Fanuc TP program (LS listing): DISTI_CADC_V16.LS

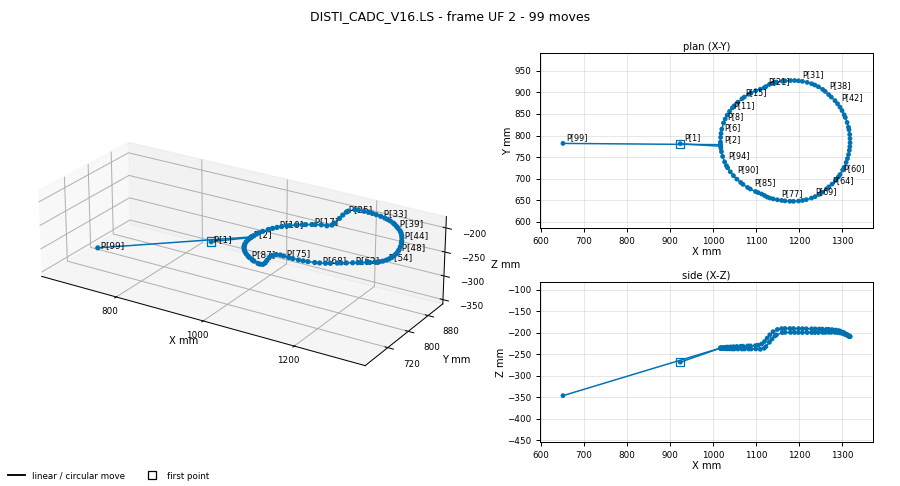
[picture p0: tool path of DISTI_CADC_V16.LS in frame UF 2, 99 of 99 moves have a stored position in this frame; points joined in program order, loops and branches not executed]
/PROG  DISTI_CADC_V16
/ATTR
OWNER		= MNEDITOR;
COMMENT		= "WeldPRO Auto-Gen";
PROG_SIZE	= 7125;
CREATE		= DATE 26-07-30  TIME 16:10:00;
MODIFIED	= DATE 26-07-30  TIME 16:41:22;
FILE_NAME	= DISTI_CA;
VERSION		= 0;
LINE_COUNT	= 113;
MEMORY_SIZE	= 7445;
PROTECT		= READ_WRITE;
TCD:  STACK_SIZE	= 0,
      TASK_PRIORITY	= 50,
      TIME_SLICE	= 0,
      BUSY_LAMP_OFF	= 0,
      ABORT_REQUEST	= 0,
      PAUSE_REQUEST	= 0;
DEFAULT_GROUP	= 1,*,*,*,*;
CONTROL_CODE	= 00000000 00000000;
/APPL
/MN
   1:  !WeldPRO Auto-Generated TPP ;
   2:  !TOR_XL_2026, TOR_xl_2907 ;
   3:   ;
   4:  UFRAME_NUM=2 ;
   5:  UTOOL_NUM=2 ;
   6:  !Feature Approach ;
   7:J P[1] 100% FINE    ;
   8:   ;
   9:  !Segment1 ;
  10:L P[2] 2000mm/sec FINE    ;
  11:   ;
  12:  CALL LASER_OFF    ;
  13:L P[3] R[23:moving]mm/sec CNT100    ;
  14:L P[4] R[23:moving]mm/sec CNT100    ;
  15:L P[5] R[23:moving]mm/sec CNT100    ;
  16:L P[6] R[23:moving]mm/sec CNT100    ;
  17:L P[7] R[23:moving]mm/sec CNT100    ;
  18:L P[8] R[23:moving]mm/sec CNT100    ;
  19:L P[9] R[23:moving]mm/sec CNT100    ;
  20:L P[10] R[23:moving]mm/sec CNT100    ;
  21:L P[11] R[23:moving]mm/sec CNT100    ;
  22:L P[12] R[23:moving]mm/sec CNT100    ;
  23:L P[13] R[23:moving]mm/sec CNT100    ;
  24:L P[14] R[23:moving]mm/sec CNT100    ;
  25:L P[15] R[23:moving]mm/sec CNT100    ;
  26:L P[16] R[23:moving]mm/sec CNT100    ;
  27:L P[17] R[23:moving]mm/sec CNT100    ;
  28:L P[18] R[23:moving]mm/sec CNT100    ;
  29:L P[19] R[23:moving]mm/sec CNT100    ;
  30:L P[20] R[23:moving]mm/sec CNT100    ;
  31:L P[21] R[23:moving]mm/sec CNT100    ;
  32:L P[22] R[23:moving]mm/sec CNT100    ;
  33:L P[23] R[23:moving]mm/sec CNT100    ;
  34:L P[24] R[23:moving]mm/sec CNT100    ;
  35:L P[25] R[23:moving]mm/sec CNT100    ;
  36:L P[26] R[23:moving]mm/sec CNT100    ;
  37:L P[27] R[23:moving]mm/sec CNT100    ;
  38:L P[28] R[23:moving]mm/sec CNT100    ;
  39:L P[29] R[23:moving]mm/sec CNT100    ;
  40:L P[30] R[23:moving]mm/sec CNT100    ;
  41:L P[31] R[23:moving]mm/sec CNT100    ;
  42:L P[32] R[23:moving]mm/sec CNT100    ;
  43:L P[33] R[23:moving]mm/sec CNT100    ;
  44:L P[34] R[23:moving]mm/sec CNT100    ;
  45:L P[35] R[23:moving]mm/sec CNT100    ;
  46:L P[36] R[23:moving]mm/sec CNT100    ;
  47:L P[37] R[23:moving]mm/sec CNT100    ;
  48:L P[38] R[23:moving]mm/sec CNT100    ;
  49:L P[39] R[23:moving]mm/sec CNT100    ;
  50:L P[40] R[23:moving]mm/sec CNT100    ;
  51:L P[41] R[23:moving]mm/sec CNT100    ;
  52:L P[42] R[23:moving]mm/sec CNT100    ;
  53:L P[43] R[23:moving]mm/sec CNT100    ;
  54:L P[44] R[23:moving]mm/sec CNT100    ;
  55:L P[45] R[23:moving]mm/sec CNT100    ;
  56:L P[46] R[23:moving]mm/sec CNT100    ;
  57:L P[47] R[23:moving]mm/sec CNT100    ;
  58:L P[48] R[23:moving]mm/sec CNT100    ;
  59:L P[49] R[23:moving]mm/sec CNT100    ;
  60:L P[50] R[23:moving]mm/sec CNT100    ;
  61:L P[51] R[23:moving]mm/sec CNT100    ;
  62:L P[52] R[23:moving]mm/sec CNT100    ;
  63:L P[53] R[23:moving]mm/sec CNT100    ;
  64:L P[54] R[23:moving]mm/sec CNT100    ;
  65:L P[55] R[23:moving]mm/sec CNT100    ;
  66:L P[56] R[23:moving]mm/sec CNT100    ;
  67:L P[57] R[23:moving]mm/sec CNT100    ;
  68:L P[58] R[23:moving]mm/sec CNT100    ;
  69:L P[59] R[23:moving]mm/sec CNT100    ;
  70:L P[60] R[23:moving]mm/sec CNT100    ;
  71:L P[61] R[23:moving]mm/sec CNT100    ;
  72:L P[62] R[23:moving]mm/sec CNT100    ;
  73:L P[63] R[23:moving]mm/sec CNT100    ;
  74:L P[64] R[23:moving]mm/sec CNT100    ;
  75:L P[65] R[23:moving]mm/sec CNT100    ;
  76:L P[66] R[23:moving]mm/sec CNT100    ;
  77:L P[67] R[23:moving]mm/sec CNT100    ;
  78:L P[68] R[23:moving]mm/sec CNT100    ;
  79:L P[69] R[23:moving]mm/sec CNT100    ;
  80:L P[70] R[23:moving]mm/sec CNT100    ;
  81:L P[71] R[23:moving]mm/sec CNT100    ;
  82:L P[72] R[23:moving]mm/sec CNT100    ;
  83:L P[73] R[23:moving]mm/sec CNT100    ;
  84:L P[74] R[23:moving]mm/sec CNT100    ;
  85:L P[75] R[23:moving]mm/sec CNT100    ;
  86:L P[76] R[23:moving]mm/sec CNT100    ;
  87:L P[77] R[23:moving]mm/sec CNT100    ;
  88:L P[78] R[23:moving]mm/sec CNT100    ;
  89:L P[79] R[23:moving]mm/sec CNT100    ;
  90:L P[80] R[23:moving]mm/sec CNT100    ;
  91:L P[81] R[23:moving]mm/sec CNT100    ;
  92:L P[82] R[23:moving]mm/sec CNT100    ;
  93:L P[83] R[23:moving]mm/sec CNT100    ;
  94:L P[84] R[23:moving]mm/sec CNT100    ;
  95:L P[85] R[23:moving]mm/sec CNT100    ;
  96:L P[86] R[23:moving]mm/sec CNT100    ;
  97:L P[87] R[23:moving]mm/sec CNT100    ;
  98:L P[88] R[23:moving]mm/sec CNT100    ;
  99:L P[89] R[23:moving]mm/sec CNT100    ;
 100:L P[90] R[23:moving]mm/sec CNT100    ;
 101:L P[91] R[23:moving]mm/sec CNT100    ;
 102:L P[92] R[23:moving]mm/sec CNT100    ;
 103:L P[93] R[23:moving]mm/sec CNT100    ;
 104:L P[94] R[23:moving]mm/sec CNT100    ;
 105:L P[95] R[23:moving]mm/sec CNT100    ;
 106:L P[96] R[23:moving]mm/sec CNT100    ;
 107:L P[97] R[23:moving]mm/sec CNT100    ;
 108:L P[98] R[23:moving]mm/sec FINE    ;
 109:  CALL LASER_OFF    ;
 110:   ;
 111:  !Feature Retreat ;
 112:L P[99] 2000mm/sec FINE    ;
 113:  CALL ROTATE    ;
/POS
P[1]{
   GP1:
	UF : 2, UT : 2,		CONFIG : 'F D T, 0, 0, 0',
	X =   924.335  mm,	Y =   780.986  mm,	Z =  -268.284  mm,
	W =  -106.495 deg,	P =   -15.000 deg,	R =    94.234 deg
};
P[2]{
   GP1:
	UF : 2, UT : 2,		CONFIG : 'F D T, 0, 0, 0',
	X =  1018.056  mm,	Y =   775.023  mm,	Z =  -235.341  mm,
	W =  -106.497 deg,	P =   -14.995 deg,	R =    94.216 deg
};
P[3]{
   GP1:
	UF : 2, UT : 2,		CONFIG : 'F D T, 0, 0, 0',
	X =  1017.747  mm,	Y =   778.750  mm,	Z =  -235.476  mm,
	W =  -106.499 deg,	P =   -14.997 deg,	R =    94.226 deg
};
P[4]{
   GP1:
	UF : 2, UT : 2,		CONFIG : 'F D T, 0, 0, 0',
	X =  1017.529  mm,	Y =   784.885  mm,	Z =  -235.671  mm,
	W =  -106.492 deg,	P =   -15.098 deg,	R =    90.372 deg
};
P[5]{
   GP1:
	UF : 2, UT : 2,		CONFIG : 'F D T, 0, 0, 0',
	X =  1017.822  mm,	Y =   795.677  mm,	Z =  -236.023  mm,
	W =  -106.481 deg,	P =   -15.218 deg,	R =    85.605 deg
};
P[6]{
   GP1:
	UF : 2, UT : 2,		CONFIG : 'F D T, 0, 0, 0',
	X =  1018.769  mm,	Y =   804.737  mm,	Z =  -236.294  mm,
	W =  -106.456 deg,	P =   -15.335 deg,	R =    80.815 deg
};
P[7]{
   GP1:
	UF : 2, UT : 2,		CONFIG : 'F D T, 0, 0, 0',
	X =  1020.603  mm,	Y =   814.889  mm,	Z =  -236.584  mm,
	W =  -106.423 deg,	P =   -15.450 deg,	R =    76.090 deg
};
P[8]{
   GP1:
	UF : 2, UT : 2,		CONFIG : 'F D T, 0, 0, 0',
	X =  1024.706  mm,	Y =   829.087  mm,	Z =  -236.960  mm,
	W =  -106.378 deg,	P =   -15.565 deg,	R =    71.217 deg
};
P[9]{
   GP1:
	UF : 2, UT : 2,		CONFIG : 'F D T, 0, 0, 0',
	X =  1028.541  mm,	Y =   838.369  mm,	Z =  -237.167  mm,
	W =  -106.322 deg,	P =   -15.679 deg,	R =    66.207 deg
};
P[10]{
   GP1:
	UF : 2, UT : 2,		CONFIG : 'F D T, 0, 0, 0',
	X =  1033.199  mm,	Y =   847.296  mm,	Z =  -237.341  mm,
	W =  -106.254 deg,	P =   -15.791 deg,	R =    61.015 deg
};
P[11]{
   GP1:
	UF : 2, UT : 2,		CONFIG : 'F D T, 0, 0, 0',
	X =  1038.649  mm,	Y =   855.813  mm,	Z =  -237.480  mm,
	W =  -106.177 deg,	P =   -15.894 deg,	R =    55.979 deg
};
P[12]{
   GP1:
	UF : 2, UT : 2,		CONFIG : 'F D T, 0, 0, 0',
	X =  1045.212  mm,	Y =   864.317  mm,	Z =  -237.594  mm,
	W =  -106.096 deg,	P =   -15.986 deg,	R =    51.162 deg
};
P[13]{
   GP1:
	UF : 2, UT : 2,		CONFIG : 'F D T, 0, 0, 0',
	X =  1049.371  mm,	Y =   868.968  mm,	Z =  -237.634  mm,
	W =  -106.012 deg,	P =   -16.066 deg,	R =    46.632 deg
};
P[14]{
   GP1:
	UF : 2, UT : 2,		CONFIG : 'F D T, 0, 0, 0',
	X =  1057.983  mm,	Y =   877.408  mm,	Z =  -237.696  mm,
	W =  -105.919 deg,	P =   -16.142 deg,	R =    41.952 deg
};
P[15]{
   GP1:
	UF : 2, UT : 2,		CONFIG : 'F D T, 0, 0, 0',
	X =  1067.342  mm,	Y =   885.184  mm,	Z =  -237.726  mm,
	W =  -105.870 deg,	P =   -16.177 deg,	R =    39.609 deg
};
P[16]{
   GP1:
	UF : 2, UT : 2,		CONFIG : 'F D T, 0, 0, 0',
	X =  1072.846  mm,	Y =   889.199  mm,	Z =  -237.714  mm,
	W =  -105.777 deg,	P =   -16.235 deg,	R =    35.365 deg
};
P[17]{
   GP1:
	UF : 2, UT : 2,		CONFIG : 'F D T, 0, 0, 0',
	X =  1083.076  mm,	Y =   895.753  mm,	Z =  -237.672  mm,
	W =  -105.677 deg,	P =   -16.289 deg,	R =    30.964 deg
};
P[18]{
   GP1:
	UF : 2, UT : 2,		CONFIG : 'F D T, 0, 0, 0',
	X =  1088.699  mm,	Y =   898.833  mm,	Z =  -237.626  mm,
	W =  -105.579 deg,	P =   -16.333 deg,	R =    26.830 deg
};
P[19]{
   GP1:
	UF : 2, UT : 2,		CONFIG : 'F D T, 0, 0, 0',
	X =  1099.375  mm,	Y =   903.910  mm,	Z =  -237.529  mm,
	W =  -105.537 deg,	P =   -16.344 deg,	R =    25.018 deg
};
P[20]{
   GP1:
	UF : 2, UT : 2,		CONFIG : 'F D T, 0, 0, 0',
	X =  1109.935  mm,	Y =   907.416  mm,	Z =  -238.388  mm,
	W =  -116.027 deg,	P =   -16.063 deg,	R =    30.267 deg
};
P[21]{
   GP1:
	UF : 2, UT : 2,		CONFIG : 'F D T, 0, 0, 0',
	X =  1119.155  mm,	Y =   910.691  mm,	Z =  -235.995  mm,
	W =  -126.877 deg,	P =   -15.356 deg,	R =    25.893 deg
};
P[22]{
   GP1:
	UF : 2, UT : 2,		CONFIG : 'F D T, 0, 0, 0',
	X =  1123.069  mm,	Y =   913.523  mm,	Z =  -231.973  mm,
	W =  -119.393 deg,	P =   -15.981 deg,	R =    16.221 deg
};
P[23]{
   GP1:
	UF : 2, UT : 2,		CONFIG : 'F D T, 0, 0, 0',
	X =  1131.162  mm,	Y =   918.546  mm,	Z =  -222.047  mm,
	W =  -115.329 deg,	P =   -16.208 deg,	R =    11.788 deg
};
P[24]{
   GP1:
	UF : 2, UT : 2,		CONFIG : 'F D T, 0, 0, 0',
	X =  1137.116  mm,	Y =   920.955  mm,	Z =  -214.516  mm,
	W =  -112.639 deg,	P =   -16.315 deg,	R =     9.714 deg
};
P[25]{
   GP1:
	UF : 2, UT : 2,		CONFIG : 'F D T, 0, 0, 0',
	X =  1143.743  mm,	Y =   923.008  mm,	Z =  -207.593  mm,
	W =  -110.015 deg,	P =   -16.386 deg,	R =     9.649 deg
};
P[26]{
   GP1:
	UF : 2, UT : 2,		CONFIG : 'F D T, 0, 0, 0',
	X =  1147.314  mm,	Y =   923.868  mm,	Z =  -205.008  mm,
	W =  -108.552 deg,	P =   -16.418 deg,	R =     8.950 deg
};
P[27]{
   GP1:
	UF : 2, UT : 2,		CONFIG : 'F D T, 0, 0, 0',
	X =  1161.002  mm,	Y =   926.134  mm,	Z =  -199.685  mm,
	W =  -105.409 deg,	P =   -16.443 deg,	R =     6.805 deg
};
P[28]{
   GP1:
	UF : 2, UT : 2,		CONFIG : 'F D T, 0, 0, 0',
	X =  1167.566  mm,	Y =   926.818  mm,	Z =  -199.138  mm,
	W =  -104.866 deg,	P =   -16.444 deg,	R =     5.597 deg
};
P[29]{
   GP1:
	UF : 2, UT : 2,		CONFIG : 'F D T, 0, 0, 0',
	X =  1180.133  mm,	Y =   927.594  mm,	Z =  -199.280  mm,
	W =  -104.887 deg,	P =   -16.444 deg,	R =     3.523 deg
};
P[30]{
   GP1:
	UF : 2, UT : 2,		CONFIG : 'F D T, 0, 0, 0',
	X =  1189.560  mm,	Y =   927.622  mm,	Z =  -199.368  mm,
	W =  -104.930 deg,	P =   -16.439 deg,	R =     -.729 deg
};
P[31]{
   GP1:
	UF : 2, UT : 2,		CONFIG : 'F D T, 0, 0, 0',
	X =  1198.430  mm,	Y =   927.043  mm,	Z =  -199.432  mm,
	W =  -104.979 deg,	P =   -16.424 deg,	R =    -5.541 deg
};
P[32]{
   GP1:
	UF : 2, UT : 2,		CONFIG : 'F D T, 0, 0, 0',
	X =  1207.671  mm,	Y =   925.761  mm,	Z =  -199.478  mm,
	W =  -105.028 deg,	P =   -16.400 deg,	R =   -10.259 deg
};
P[33]{
   GP1:
	UF : 2, UT : 2,		CONFIG : 'F D T, 0, 0, 0',
	X =  1218.717  mm,	Y =   923.312  mm,	Z =  -199.499  mm,
	W =  -105.070 deg,	P =   -16.371 deg,	R =   -14.490 deg
};
P[34]{
   GP1:
	UF : 2, UT : 2,		CONFIG : 'F D T, 0, 0, 0',
	X =  1229.164  mm,	Y =   920.085  mm,	Z =  -199.490  mm,
	W =  -105.112 deg,	P =   -16.334 deg,	R =   -18.515 deg
};
P[35]{
   GP1:
	UF : 2, UT : 2,		CONFIG : 'F D T, 0, 0, 0',
	X =  1236.746  mm,	Y =   917.127  mm,	Z =  -199.468  mm,
	W =  -105.158 deg,	P =   -16.285 deg,	R =   -23.051 deg
};
P[36]{
   GP1:
	UF : 2, UT : 2,		CONFIG : 'F D T, 0, 0, 0',
	X =  1244.915  mm,	Y =   913.195  mm,	Z =  -199.425  mm,
	W =  -105.219 deg,	P =   -16.204 deg,	R =   -29.417 deg
};
P[37]{
   GP1:
	UF : 2, UT : 2,		CONFIG : 'F D T, 0, 0, 0',
	X =  1254.809  mm,	Y =   906.969  mm,	Z =  -199.336  mm,
	W =  -105.311 deg,	P =   -16.047 deg,	R =   -39.415 deg
};
P[38]{
   GP1:
	UF : 2, UT : 2,		CONFIG : 'F D T, 0, 0, 0',
	X =  1260.595  mm,	Y =   902.395  mm,	Z =  -199.225  mm,
	W =  -105.307 deg,	P =   -16.055 deg,	R =   -38.974 deg
};
P[39]{
   GP1:
	UF : 2, UT : 2,		CONFIG : 'F D T, 0, 0, 0',
	X =  1268.689  mm,	Y =   894.946  mm,	Z =  -199.033  mm,
	W =  -105.302 deg,	P =   -16.063 deg,	R =   -38.625 deg
};
P[40]{
   GP1:
	UF : 2, UT : 2,		CONFIG : 'F D T, 0, 0, 0',
	X =  1274.754  mm,	Y =   889.208  mm,	Z =  -198.997  mm,
	W =  -105.469 deg,	P =   -15.944 deg,	R =   -44.976 deg
};
P[41]{
   GP1:
	UF : 2, UT : 2,		CONFIG : 'F D T, 0, 0, 0',
	X =  1283.308  mm,	Y =   880.882  mm,	Z =  -199.181  mm,
	W =  -105.661 deg,	P =   -15.890 deg,	R =   -47.714 deg
};
P[42]{
   GP1:
	UF : 2, UT : 2,		CONFIG : 'F D T, 0, 0, 0',
	X =  1289.303  mm,	Y =   873.818  mm,	Z =  -199.609  mm,
	W =  -106.210 deg,	P =   -15.792 deg,	R =   -52.259 deg
};
P[43]{
   GP1:
	UF : 2, UT : 2,		CONFIG : 'F D T, 0, 0, 0',
	X =  1294.880  mm,	Y =   865.895  mm,	Z =  -200.330  mm,
	W =  -106.927 deg,	P =   -15.688 deg,	R =   -56.663 deg
};
P[44]{
   GP1:
	UF : 2, UT : 2,		CONFIG : 'F D T, 0, 0, 0',
	X =  1299.661  mm,	Y =   857.908  mm,	Z =  -201.305  mm,
	W =  -107.603 deg,	P =   -15.597 deg,	R =   -60.243 deg
};
P[45]{
   GP1:
	UF : 2, UT : 2,		CONFIG : 'F D T, 0, 0, 0',
	X =  1304.641  mm,	Y =   848.096  mm,	Z =  -202.841  mm,
	W =  -108.271 deg,	P =   -15.504 deg,	R =   -63.685 deg
};
P[46]{
   GP1:
	UF : 2, UT : 2,		CONFIG : 'F D T, 0, 0, 0',
	X =  1307.301  mm,	Y =   841.848  mm,	Z =  -204.015  mm,
	W =  -109.144 deg,	P =   -15.377 deg,	R =   -68.203 deg
};
P[47]{
   GP1:
	UF : 2, UT : 2,		CONFIG : 'F D T, 0, 0, 0',
	X =  1311.509  mm,	Y =   830.300  mm,	Z =  -206.050  mm,
	W =  -109.899 deg,	P =   -15.253 deg,	R =   -72.505 deg
};
P[48]{
   GP1:
	UF : 2, UT : 2,		CONFIG : 'F D T, 0, 0, 0',
	X =  1314.580  mm,	Y =   819.354  mm,	Z =  -207.483  mm,
	W =  -110.273 deg,	P =   -15.181 deg,	R =   -74.981 deg
};
P[49]{
   GP1:
	UF : 2, UT : 2,		CONFIG : 'F D T, 0, 0, 0',
	X =  1315.840  mm,	Y =   813.364  mm,	Z =  -208.079  mm,
	W =  -110.635 deg,	P =   -14.305 deg,	R =   -78.232 deg
};
P[50]{
   GP1:
	UF : 2, UT : 2,		CONFIG : 'F D T, 0, 0, 0',
	X =  1317.453  mm,	Y =   802.522  mm,	Z =  -208.765  mm,
	W =  -111.054 deg,	P =   -14.769 deg,	R =   -83.164 deg
};
P[51]{
   GP1:
	UF : 2, UT : 2,		CONFIG : 'F D T, 0, 0, 0',
	X =  1318.169  mm,	Y =   792.882  mm,	Z =  -208.974  mm,
	W =  -111.190 deg,	P =   -15.305 deg,	R =   -88.308 deg
};
P[52]{
   GP1:
	UF : 2, UT : 2,		CONFIG : 'F D T, 0, 0, 0',
	X =  1318.266  mm,	Y =   783.191  mm,	Z =  -208.811  mm,
	W =  -111.129 deg,	P =   -15.645 deg,	R =   -91.614 deg
};
P[53]{
   GP1:
	UF : 2, UT : 2,		CONFIG : 'F D T, 0, 0, 0',
	X =  1317.713  mm,	Y =   774.210  mm,	Z =  -208.329  mm,
	W =  -110.761 deg,	P =   -14.624 deg,	R =   -96.574 deg
};
P[54]{
   GP1:
	UF : 2, UT : 2,		CONFIG : 'F D T, 0, 0, 0',
	X =  1316.659  mm,	Y =   765.677  mm,	Z =  -207.557  mm,
	W =  -110.276 deg,	P =   -14.535 deg,	R =  -100.836 deg
};
P[55]{
   GP1:
	UF : 2, UT : 2,		CONFIG : 'F D T, 0, 0, 0',
	X =  1314.782  mm,	Y =   755.866  mm,	Z =  -206.306  mm,
	W =  -109.635 deg,	P =   -14.447 deg,	R =  -105.265 deg
};
P[56]{
   GP1:
	UF : 2, UT : 2,		CONFIG : 'F D T, 0, 0, 0',
	X =  1312.289  mm,	Y =   746.477  mm,	Z =  -204.738  mm,
	W =  -109.083 deg,	P =   -14.382 deg,	R =  -108.625 deg
};
P[57]{
   GP1:
	UF : 2, UT : 2,		CONFIG : 'F D T, 0, 0, 0',
	X =  1309.253  mm,	Y =   737.576  mm,	Z =  -202.914  mm,
	W =  -108.349 deg,	P =   -14.302 deg,	R =  -112.873 deg
};
P[58]{
   GP1:
	UF : 2, UT : 2,		CONFIG : 'F D T, 0, 0, 0',
	X =  1304.195  mm,	Y =   725.757  mm,	Z =  -199.953  mm,
	W =  -107.748 deg,	P =   -14.239 deg,	R =  -116.265 deg
};
P[59]{
   GP1:
	UF : 2, UT : 2,		CONFIG : 'F D T, 0, 0, 0',
	X =  1301.193  mm,	Y =   719.919  mm,	Z =  -198.437  mm,
	W =  -106.927 deg,	P =   -14.148 deg,	R =  -121.193 deg
};
P[60]{
   GP1:
	UF : 2, UT : 2,		CONFIG : 'F D T, 0, 0, 0',
	X =  1294.925  mm,	Y =   709.284  mm,	Z =  -196.020  mm,
	W =  -106.269 deg,	P =   -14.066 deg,	R =  -125.698 deg
};
P[61]{
   GP1:
	UF : 2, UT : 2,		CONFIG : 'F D T, 0, 0, 0',
	X =  1291.201  mm,	Y =   703.877  mm,	Z =  -195.000  mm,
	W =  -105.781 deg,	P =   -13.988 deg,	R =  -130.143 deg
};
P[62]{
   GP1:
	UF : 2, UT : 2,		CONFIG : 'F D T, 0, 0, 0',
	X =  1284.891  mm,	Y =   695.831  mm,	Z =  -193.723  mm,
	W =  -105.527 deg,	P =   -13.913 deg,	R =  -134.519 deg
};
P[63]{
   GP1:
	UF : 2, UT : 2,		CONFIG : 'F D T, 0, 0, 0',
	X =  1276.648  mm,	Y =   687.317  mm,	Z =  -192.688  mm,
	W =  -105.437 deg,	P =   -13.849 deg,	R =  -138.629 deg
};
P[64]{
   GP1:
	UF : 2, UT : 2,		CONFIG : 'F D T, 0, 0, 0',
	X =  1269.179  mm,	Y =   680.825  mm,	Z =  -192.113  mm,
	W =  -105.429 deg,	P =   -13.831 deg,	R =  -139.837 deg
};
P[65]{
   GP1:
	UF : 2, UT : 2,		CONFIG : 'F D T, 0, 0, 0',
	X =  1263.935  mm,	Y =   676.312  mm,	Z =  -191.836  mm,
	W =  -105.443 deg,	P =   -13.863 deg,	R =  -137.727 deg
};
P[66]{
   GP1:
	UF : 2, UT : 2,		CONFIG : 'F D T, 0, 0, 0',
	X =  1254.091  mm,	Y =   668.195  mm,	Z =  -191.502  mm,
	W =  -105.373 deg,	P =   -13.729 deg,	R =  -147.436 deg
};
P[67]{
   GP1:
	UF : 2, UT : 2,		CONFIG : 'F D T, 0, 0, 0',
	X =  1246.737  mm,	Y =   663.238  mm,	Z =  -191.280  mm,
	W =  -105.298 deg,	P =   -13.637 deg,	R =  -156.529 deg
};
P[68]{
   GP1:
	UF : 2, UT : 2,		CONFIG : 'F D T, 0, 0, 0',
	X =  1237.336  mm,	Y =   658.201  mm,	Z =  -191.018  mm,
	W =  -105.277 deg,	P =   -13.618 deg,	R =  -158.976 deg
};
P[69]{
   GP1:
	UF : 2, UT : 2,		CONFIG : 'F D T, 0, 0, 0',
	X =  1228.976  mm,	Y =   654.840  mm,	Z =  -190.829  mm,
	W =  -105.241 deg,	P =   -13.592 deg,	R =  -162.969 deg
};
P[70]{
   GP1:
	UF : 2, UT : 2,		CONFIG : 'F D T, 0, 0, 0',
	X =  1216.767  mm,	Y =   651.155  mm,	Z =  -190.593  mm,
	W =  -105.203 deg,	P =   -13.573 deg,	R =  -167.022 deg
};
P[71]{
   GP1:
	UF : 2, UT : 2,		CONFIG : 'F D T, 0, 0, 0',
	X =  1207.937  mm,	Y =   649.248  mm,	Z =  -190.450  mm,
	W =  -105.159 deg,	P =   -13.560 deg,	R =  -171.569 deg
};
P[72]{
   GP1:
	UF : 2, UT : 2,		CONFIG : 'F D T, 0, 0, 0',
	X =  1198.766  mm,	Y =   647.917  mm,	Z =  -190.323  mm,
	W =  -105.113 deg,	P =   -13.556 deg,	R =  -176.312 deg
};
P[73]{
   GP1:
	UF : 2, UT : 2,		CONFIG : 'F D T, 0, 0, 0',
	X =  1187.063  mm,	Y =   647.196  mm,	Z =  -190.190  mm,
	W =  -105.068 deg,	P =   -13.561 deg,	R =   179.213 deg
};
P[74]{
   GP1:
	UF : 2, UT : 2,		CONFIG : 'F D T, 0, 0, 0',
	X =  1178.653  mm,	Y =   647.351  mm,	Z =  -190.117  mm,
	W =  -105.038 deg,	P =   -13.569 deg,	R =   176.231 deg
};
P[75]{
   GP1:
	UF : 2, UT : 2,		CONFIG : 'F D T, 0, 0, 0',
	X =  1167.247  mm,	Y =   648.254  mm,	Z =  -190.073  mm,
	W =  -105.207 deg,	P =   -13.572 deg,	R =   175.290 deg
};
P[76]{
   GP1:
	UF : 2, UT : 2,		CONFIG : 'F D T, 0, 0, 0',
	X =  1159.511  mm,	Y =   649.280  mm,	Z =  -190.357  mm,
	W =  -107.012 deg,	P =   -13.569 deg,	R =   174.537 deg
};
P[77]{
   GP1:
	UF : 2, UT : 2,		CONFIG : 'F D T, 0, 0, 0',
	X =  1149.633  mm,	Y =   650.867  mm,	Z =  -192.370  mm,
	W =  -109.414 deg,	P =   -13.538 deg,	R =   174.483 deg
};
P[78]{
   GP1:
	UF : 2, UT : 2,		CONFIG : 'F D T, 0, 0, 0',
	X =  1139.791  mm,	Y =   652.860  mm,	Z =  -197.490  mm,
	W =  -112.196 deg,	P =   -13.466 deg,	R =   175.323 deg
};
P[79]{
   GP1:
	UF : 2, UT : 2,		CONFIG : 'F D T, 0, 0, 0',
	X =  1132.005  mm,	Y =   654.923  mm,	Z =  -204.720  mm,
	W =  -114.872 deg,	P =   -13.369 deg,	R =   175.422 deg
};
P[80]{
   GP1:
	UF : 2, UT : 2,		CONFIG : 'F D T, 0, 0, 0',
	X =  1125.887  mm,	Y =   657.208  mm,	Z =  -212.500  mm,
	W =  -120.114 deg,	P =   -13.109 deg,	R =   172.293 deg
};
P[81]{
   GP1:
	UF : 2, UT : 2,		CONFIG : 'F D T, 0, 0, 0',
	X =  1119.872  mm,	Y =   660.702  mm,	Z =  -220.322  mm,
	W =  -126.810 deg,	P =   -12.622 deg,	R =   167.787 deg
};
P[82]{
   GP1:
	UF : 2, UT : 2,		CONFIG : 'F D T, 0, 0, 0',
	X =  1112.921  mm,	Y =   664.265  mm,	Z =  -226.144  mm,
	W =  -119.561 deg,	P =   -13.285 deg,	R =   157.806 deg
};
P[83]{
   GP1:
	UF : 2, UT : 2,		CONFIG : 'F D T, 0, 0, 0',
	X =  1104.974  mm,	Y =   667.456  mm,	Z =  -228.841  mm,
	W =  -107.219 deg,	P =   -13.741 deg,	R =   154.408 deg
};
P[84]{
   GP1:
	UF : 2, UT : 2,		CONFIG : 'F D T, 0, 0, 0',
	X =  1098.910  mm,	Y =   669.923  mm,	Z =  -229.763  mm,
	W =  -105.746 deg,	P =   -13.749 deg,	R =   154.142 deg
};
P[85]{
   GP1:
	UF : 2, UT : 2,		CONFIG : 'F D T, 0, 0, 0',
	X =  1086.709  mm,	Y =   675.819  mm,	Z =  -230.299  mm,
	W =  -105.804 deg,	P =   -13.784 deg,	R =   151.506 deg
};
P[86]{
   GP1:
	UF : 2, UT : 2,		CONFIG : 'F D T, 0, 0, 0',
	X =  1080.683  mm,	Y =   679.329  mm,	Z =  -230.577  mm,
	W =  -105.885 deg,	P =   -13.838 deg,	R =   147.739 deg
};
P[87]{
   GP1:
	UF : 2, UT : 2,		CONFIG : 'F D T, 0, 0, 0',
	X =  1069.857  mm,	Y =   686.687  mm,	Z =  -231.107  mm,
	W =  -105.988 deg,	P =   -13.918 deg,	R =   142.681 deg
};
P[88]{
   GP1:
	UF : 2, UT : 2,		CONFIG : 'F D T, 0, 0, 0',
	X =  1064.555  mm,	Y =   690.903  mm,	Z =  -231.378  mm,
	W =  -106.082 deg,	P =   -14.006 deg,	R =   137.688 deg
};
P[89]{
   GP1:
	UF : 2, UT : 2,		CONFIG : 'F D T, 0, 0, 0',
	X =  1055.598  mm,	Y =   698.727  mm,	Z =  -231.835  mm,
	W =  -106.129 deg,	P =   -14.056 deg,	R =   135.015 deg
};
P[90]{
   GP1:
	UF : 2, UT : 2,		CONFIG : 'F D T, 0, 0, 0',
	X =  1047.587  mm,	Y =   706.947  mm,	Z =  -232.297  mm,
	W =  -106.186 deg,	P =   -14.117 deg,	R =   131.622 deg
};
P[91]{
   GP1:
	UF : 2, UT : 2,		CONFIG : 'F D T, 0, 0, 0',
	X =  1040.435  mm,	Y =   715.740  mm,	Z =  -232.796  mm,
	W =  -106.269 deg,	P =   -14.239 deg,	R =   125.999 deg
};
P[92]{
   GP1:
	UF : 2, UT : 2,		CONFIG : 'F D T, 0, 0, 0',
	X =  1034.147  mm,	Y =   725.125  mm,	Z =  -233.271  mm,
	W =  -106.343 deg,	P =   -14.367 deg,	R =   120.225 deg
};
P[93]{
   GP1:
	UF : 2, UT : 2,		CONFIG : 'F D T, 0, 0, 0',
	X =  1031.382  mm,	Y =   730.028  mm,	Z =  -233.484  mm,
	W =  -106.384 deg,	P =   -14.458 deg,	R =   116.261 deg
};
P[94]{
   GP1:
	UF : 2, UT : 2,		CONFIG : 'F D T, 0, 0, 0',
	X =  1027.140  mm,	Y =   738.791  mm,	Z =  -233.861  mm,
	W =  -106.433 deg,	P =   -14.556 deg,	R =   111.957 deg
};
P[95]{
   GP1:
	UF : 2, UT : 2,		CONFIG : 'F D T, 0, 0, 0',
	X =  1022.544  mm,	Y =   751.435  mm,	Z =  -234.403  mm,
	W =  -106.465 deg,	P =   -14.714 deg,	R =   105.666 deg
};
P[96]{
   GP1:
	UF : 2, UT : 2,		CONFIG : 'F D T, 0, 1, 0',
	X =  1019.785  mm,	Y =   762.599  mm,	Z =  -234.899  mm,
	W =  -106.480 deg,	P =   -14.798 deg,	R =   102.262 deg
};
P[97]{
   GP1:
	UF : 2, UT : 2,		CONFIG : 'F D T, 0, 1, 0',
	X =  1018.490  mm,	Y =   770.878  mm,	Z =  -235.202  mm,
	W =  -106.494 deg,	P =   -14.935 deg,	R =    96.827 deg
};
P[98]{
   GP1:
	UF : 2, UT : 2,		CONFIG : 'F D T, 0, 1, 0',
	X =  1017.748  mm,	Y =   778.749  mm,	Z =  -235.476  mm,
	W =  -106.501 deg,	P =   -14.999 deg,	R =    94.236 deg
};
P[99]{
   GP1:
	UF : 2, UT : 2,		CONFIG : 'F D T, 0, 1, 0',
	X =   651.995  mm,	Y =   781.694  mm,	Z =  -345.952  mm,
	W =  -106.495 deg,	P =   -15.000 deg,	R =    94.234 deg
};
/END
